Fanuc KAREL source: kt00110.KL

PROGRAM KT00110
%NOLOCKGROUP
VAR
R1:REAL
Y2 : ARRAY[2] OF BYTE
OUT:REAL
BEGIN
R1=2.0
Y2[1]=3
OUT=(R1/(Y2[1]))
END KT00110
